FUNCTION_BLOCK AX_T_FF_SR_GATE (* Wie AX_T_FF_SR, zusaetzlich mit Freigabe-Socket GATE:AX und eigenem Zustand GATE_CLOSED - ohne Verkettung (kein CHAIN_IN/CHAIN_OUT) *)
  (* Standard: 61499-1 Annex A; Function: Wie AX_T_FF_SR (lokales S/R/CLK), zusaetzlich: GATE (Socket, AX) muss TRUE sein, sonst wird der Baustein in einen eigenen Zustand GATE_CLOSED gezwungen (Q.E1 mit FALSE). In GATE_CLOSED ist S/R/CLK komplett wirkungslos (keine Transition definiert - IEC 61499 verwirft das Event einfach) - der EINZIGE Ausweg ist GATE.E1[GATE.D1] zurueck nach RESET.; Description: Copyright (c) 2017 fortiss GmbH, HR Agrartechnik GmbH This program and the accompanying materials are made available under the terms of the Eclipse Public License 2.0 which is available at https://www.eclipse.org/legal/epl-2.0/ SPDX-License-Identifier: EPL-2.0 *)
  (* Version 1.2, 2026-09-17, Franz Höpfinger, HR Agrartechnik GmbH, Bugfix (Reihenfolge-Luecke): [NOT GATE.D1] stand in RESET/SET HINTER S/CLK - da S/CLK ohne Guard immer TRUE sind, hat IEC 61499-1 Table 1 Regel c) sie zuerst gekreuzt, die Gate-Sperre kam nie zum Zug (S/CLK haben trotz geschlossenem Gate eingeschaltet). Fix: [NOT GATE.D1] in JEDEM Zustand an erste Stelle der Deklarationsreihenfolge gesetzt - ist das Gate zu, greift die Sperre garantiert zuerst; ist es offen, ist ihr Guard FALSE, wird uebersprungen, S/CLK/R wirken normal. *)
  (* Version 1.1, 2026-09-17, Franz Höpfinger, HR Agrartechnik GmbH, Ergaenzung (Franz: 'beim Betreten von START wollen wir doch dass er gleich auf GATE_CLOSED geht, falls D1 nicht da ist, egal ob ein Event GATE.E1 gekommen ist'): zusaetzliche Epsilon-Transition START->GATE_CLOSED Condition="[NOT GATE.D1]" (ohne Event davor, wie bei AX_T_FF_INIT/AX_RS_SYM_INIT's Init-Zustand [FALSE = Q_INIT]) - wird SOFORT beim Betreten von START ausgewertet, deckt das Boot-Fenster ab (Gate schon zu, BEVOR je ein GATE.E1 gefeuert hat). Kein Duplikat zu GATE.E1[NOT GATE.D1]: die Epsilon-Variante deckt den Zustand VOR dem ersten GATE-Update ab, die event-getriggerte Variante das laufende Monitoring danach - beide zusammen noetig. *)
  (* Version 1.0, 2026-09-17, Franz Höpfinger, HR Agrartechnik GmbH, Neu (Franz: 'mach gleich noch einen AX_T_FF_SR.fbt GATE ohne die Verkettung'). Kopiert von AX_T_FF_SR, um GATE:AX-Socket + Zustand GATE_CLOSED erweitert - identisches Muster wie AX_T_FF_SR_SEQ_GATE, nur ohne CHAIN_IN/CHAIN_OUT, fuer Einsatzfaelle die nur die Gate-Sperre brauchen, keine Kettenverzoegerung. *)
  (* Version 3.0, 2025-04-14, Patrick Aigner, changed package *)
  (* Version 1.1, 2024-08-27, Franz Höpfinger, HR Agrartechnik GmbH, Copy E_SR and make this FB *)
  (* Version 1.0, 2017-09-22, Alois Zoitl, fortiss GmbH, initial API and implementation and/or initial documentation *)
  PACKAGE adapter::events::unidirectional;
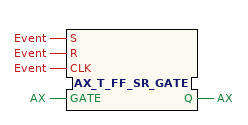
  EVENT_INPUT
    S; (* Set output Q - wirkungslos waehrend GATE_CLOSED *)
    R; (* Reset output Q - wirkungslos waehrend GATE_CLOSED (ist ohnehin schon aus) *)
    CLK; (* Clock for triggering a output toggle - wirkungslos waehrend GATE_CLOSED *)
  END_EVENT
  SOCKETS
    GATE : adapter::types::unidirectional::AX; (* Freigabe: muss TRUE sein. Faellt GATE auf FALSE: sofort GATE_CLOSED (Zwangs-RESET + Sperre), verlassen nur ueber GATE.E1[GATE.D1]. *)
  END_SOCKETS
  PLUGS
    Q : adapter::types::unidirectional::AX; (* value of flip flop *)
  END_PLUGS
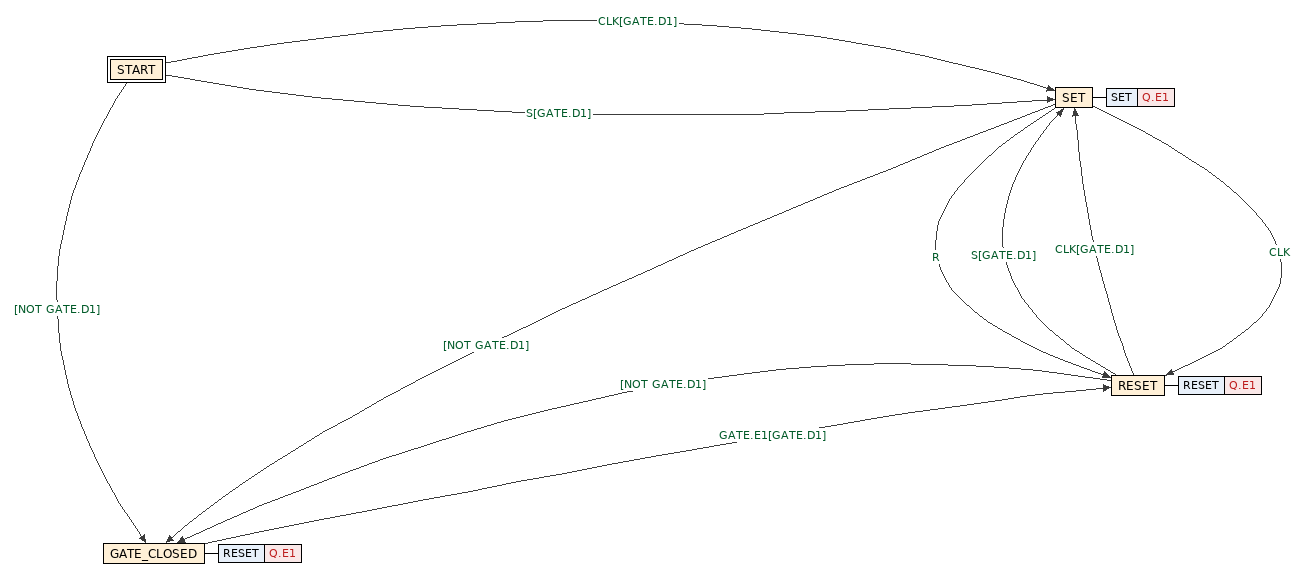
  EC_STATES
    START; (* Initial State *)
    SET : SET -> Q.E1;
    RESET : RESET -> Q.E1;
    GATE_CLOSED : RESET -> Q.E1; (* Gesperrt: GATE.D1=FALSE. Q zwangsweise FALSE. S/R/CLK sind hier wirkungslos. Einziger Ausweg: GATE.E1[GATE.D1] zurueck nach RESET. *)
  END_STATES
  EC_TRANSITIONS
    START TO GATE_CLOSED := [NOT GATE.D1];
    START TO SET := S[GATE.D1];
    START TO SET := CLK[GATE.D1];
    SET TO GATE_CLOSED := [NOT GATE.D1];
    SET TO RESET := R;
    SET TO RESET := CLK;
    RESET TO GATE_CLOSED := [NOT GATE.D1];
    RESET TO SET := S[GATE.D1];
    RESET TO SET := CLK[GATE.D1];
    GATE_CLOSED TO RESET := GATE.E1[GATE.D1];
  END_TRANSITIONS
  ALGORITHM SET IN ST:
Q.D1 := TRUE;
  END_ALGORITHM
  ALGORITHM RESET IN ST:
Q.D1 := FALSE;
  END_ALGORITHM
END_FUNCTION_BLOCK
